// TwinCAT 3 PLC project PLC_1
// ProgramVersion: 3.1.4024.0
// libraries:
//   Tc2_Standard, * (Beckhoff Automation GmbH)
//   Tc2_System, * (Beckhoff Automation GmbH)
//   Tc3_Module, * (Beckhoff Automation GmbH)
// project tree:
//   GVLs/ GVL.TcGVL
//   / PlcTask.TcTTO
//   POUs/ AnalogInputConversion.TcPOU, AnalogOutputConversion.TcPOU, InterfaceControlPanel.TcPOU, MAIN.TcPOU, ValveController.TcPOU

CONFIGURATION PLC_1
    RESOURCE PLC ON TwinCAT3
        TASK PlcTask(INTERVAL := T#10ms, PRIORITY := 20);
        PROGRAM MAIN WITH PlcTask : MAIN;
    END_RESOURCE
END_CONFIGURATION

// ---- GVLs/GVL.TcGVL
{attribute 'qualified_only'}
VAR_GLOBAL
	mb_Input_Coils : ARRAY [0..3] OF BOOL;
	mb_Output_Coils : ARRAY [0..3] OF BOOL;
	mb_Input_Registers : ARRAY [0..3] OF WORD;
	mb_Output_Registers : ARRAY [0..2] OF WORD;
END_VAR

// ---- POUs/MAIN.TcPOU
PROGRAM MAIN
VAR
	ValveController : ValveController;
	InterfaceControlPanel : InterfaceControlPanel;

	StartButton : BOOL;
	ResetButton : BOOL;
	StopButton : BOOL;
	
	StartLight : BOOL;
	ResetLight : BOOL;
	StopLight : BOOL;
	FactoryIOReset: BOOL;

	Setpoint : WORD;
	LevelMeter : WORD;
	
	FillValve : WORD;
	DischargeValve: WORD;
	SP : WORD;
	PV : WORD;
	
	SP_Scaled: REAL;
	LevelScaled: REAL;
	
	isSystemON: BOOL;
	isStopON: BOOL;
	isResetON: BOOL;
	
	tBlink: TON;
	BlinkBit: BOOL;
END_VAR

// I/O Assignments
GVL.mb_Input_Coils[0] := StartLight;
GVL.mb_Input_Coils[1] := ResetLight;
GVL.mb_Input_Coils[2] := StopLight;
GVL.mb_Input_Coils[3] := FactoryIOReset;

StartButton := GVL.mb_Output_Coils[0];
ResetButton := GVL.mb_Output_Coils[1];
StopButton := GVL.mb_Output_Coils[2];

LevelMeter := GVL.mb_Output_Registers[0];
Setpoint := GVL.mb_Output_Registers[2];

GVL.mb_Input_Registers[0] := FillValve;
GVL.mb_Input_Registers[1] := DischargeValve;
GVL.mb_Input_Registers[2] := SP;
GVL.mb_Input_Registers[3] := PV;
//
// Blink bit assignment
tBlink(IN := NOT tBlink.Q, PT := T#1000MS);
BlinkBit := tBlink.ET > T#500MS;
//
// Buttons control initialization
InterfaceControlPanel(StartButton := StartButton, ResetButton := ResetButton, StopButton := StopButton, blink := BlinkBit,
	isStopON := isStopON, isSystemON := isSystemON, isResetON := isResetON, StartLight => StartLight, StopLight => StopLight, ResetLight => ResetLight);
//
// Reset logic
IF ResetButton THEN
	FactoryIOReset := TRUE;
	isSystemON := FALSE;
	isStopON := TRUE;
ELSE
	FactoryIOReset := FALSE;
END_IF;
//
// Setpoint conversion & assignment
AnalogInputConversion(AnalogInput := Setpoint, ScaleMax := 300, ScaledValue => SP_Scaled);
SP := REAL_TO_WORD(SP_Scaled);
//
// Current water level conversion & assignment
AnalogInputConversion(AnalogInput := LevelMeter, ScaleMax := 300, ScaledValue => LevelScaled);
PV := REAL_TO_WORD(LevelScaled);
//
// Valve control logic
IF isSystemON THEN	
	IF PV < SP THEN
		AnalogOutputConversion(0.0, AnalogOutput => DischargeValve);
		ValveController(TargetWaterLevel := SP_Scaled, CurrentWaterLevel := LevelScaled, ScaleMax := 30, AnalogOutputValue => FillValve);
	END_IF;
	IF PV > SP THEN
		AnalogOutputConversion(0.0, AnalogOutput => FillValve);
		ValveController(TargetWaterLevel := LevelScaled, CurrentWaterLevel := SP_Scaled, ScaleMax := 7, AnalogOutputValue => DischargeValve);
	END_IF;
	IF PV = SP THEN
		AnalogOutputConversion(0.0, AnalogOutput => FillValve);
		AnalogOutputConversion(0.0, AnalogOutput => DischargeValve);
	END_IF;
ELSE
	AnalogOutputConversion(0.0, AnalogOutput => FillValve);
	AnalogOutputConversion(0.0, AnalogOutput => DischargeValve);
END_IF;
//

END_PROGRAM

// ---- POUs/ValveController.TcPOU
// Valve control logic (fill by default, discharge if TargetWaterLevel and CurrentWaterLevel are swapped)
FUNCTION_BLOCK PUBLIC ValveController
VAR_INPUT
	TargetWaterLevel: REAL;
	CurrentWaterLevel: REAL;
	// The value (cm) at which the flow speed will start to decrease linearly
	ScaleMax : INT;
END_VAR
VAR_OUTPUT
	AnalogOutputValue: WORD;
END_VAR
VAR
	LevelOffset : REAL;
	AnalogOutputTemp: WORD;
END_VAR

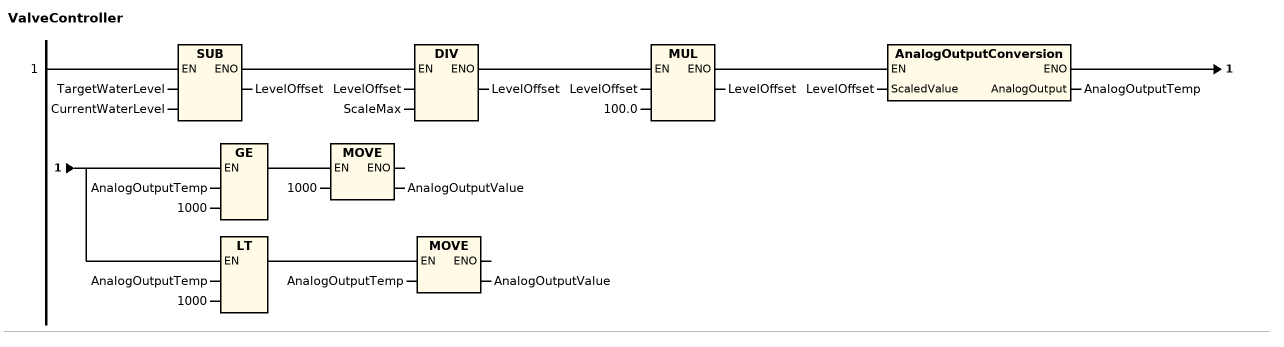
// NETWORK 1
LevelOffset := TargetWaterLevel - CurrentWaterLevel;
LevelOffset := LevelOffset / ScaleMax;
LevelOffset := LevelOffset * 100.0;
AnalogOutputConversion(ScaledValue := LevelOffset, AnalogOutput => AnalogOutputTemp);
IF AnalogOutputTemp >= 1000 THEN AnalogOutputValue := 1000; END_IF
IF AnalogOutputTemp < 1000 THEN AnalogOutputValue := AnalogOutputTemp; END_IF

END_FUNCTION_BLOCK

// ---- POUs/AnalogOutputConversion.TcPOU
// Convert normalized value to analog value
FUNCTION AnalogOutputConversion : WORD
VAR_INPUT
	ScaledValue : REAL;
END_VAR
VAR
	NormalizedValue : REAL;
END_VAR

VAR_OUTPUT
	AnalogOutput: WORD;
END_VAR

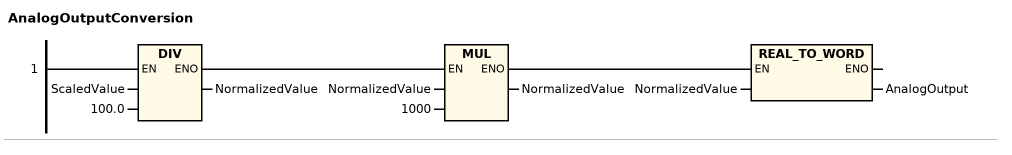
// NETWORK 1
NormalizedValue := ScaledValue / 100.0;
NormalizedValue := NormalizedValue * 1000;
AnalogOutput := REAL_TO_WORD(NormalizedValue);

END_FUNCTION

// ---- POUs/InterfaceControlPanel.TcPOU
// Buttons control logic
FUNCTION_BLOCK PUBLIC InterfaceControlPanel
VAR_INPUT
	StartButton : BOOL;
	ResetButton : BOOL;
	StopButton : BOOL;
	blink : BOOL;
END_VAR
VAR_IN_OUT
	isStopON : BOOL;
	isSystemON : BOOL;
	isResetON : BOOL;
END_VAR
VAR_OUTPUT
	StartLight : BOOL;
	StopLight : BOOL;
	ResetLight : BOOL;
END_VAR
VAR
END_VAR

// Memory bit for isSystemON
IF StartButton THEN
	isSystemON := TRUE;
END_IF;

IF NOT StopButton THEN
	isSystemON := FALSE;
END_IF;
// -------------
// Memory bit for isStopON
IF NOT StopButton THEN
	isStopON := TRUE;
END_IF;

IF isSystemON THEN
	isStopON := FALSE;
END_IF;
// -------------
// Memory bit for isResetON
IF ResetButton THEN
	isResetON := TRUE;
END_IF;

IF isSystemON THEN
	isResetON := FALSE;
END_IF;
// -------------
// ------------- OUTPUTS ---------------
StartLight := isSystemON OR (isStopON AND NOT isSystemON AND blink);
//
ResetLight := isResetON;
//
StopLight := isStopON AND NOT isSystemON;

END_FUNCTION_BLOCK

// ---- POUs/AnalogInputConversion.TcPOU
// Convert analog value to normalized value
FUNCTION AnalogInputConversion : REAL
VAR_INPUT
	// Analog Value to normalize
	AnalogInput : WORD;
	// Maximum value on the scale
	ScaleMax: INT;
END_VAR
VAR
	NormalizedInput: REAL;
END_VAR

VAR_OUTPUT
	// Normalized Output
	ScaledValue: REAL;
END_VAR

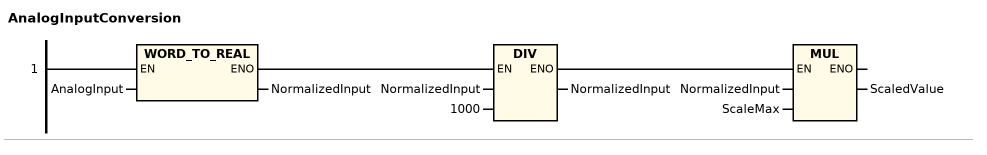
// NETWORK 1
NormalizedInput := WORD_TO_REAL(AnalogInput);
NormalizedInput := NormalizedInput / 1000;
ScaledValue := NormalizedInput * ScaleMax;

END_FUNCTION
